(* Logix 5000 project; controller Celula_Envase_Automatica Emulate 5570 rev 32.11; software revision 32.03 *)

TASK MainTask (continuous, watchdog 500 ms) : MainProgram, Sequencer, Motor, IO
TASK PID_Task (periodic, rate 100 ms, priority 10, watchdog 500 ms) : PID_Control
TASK Simulation_Task (periodic, rate 100 ms, priority 11, watchdog 500 ms) : Process_Sim

MODULES
   Local : Emulate 5570 (ICP 2, rev 32.11)
END_MODULES

TYPE UDT_Cell :
STRUCT
   Cmd_Start : BOOL;   // Comando de partida da célula
   Cmd_Stop : BOOL;   // Comando de parada da célula
   Cmd_Reset : BOOL;   // Comando de reset de falhas
   AutoMode : BOOL;   // Seleção de modo automático
   Ready : BOOL;   // Célula pronta para operar
   Running : BOOL;   // Célula em operação
   Faulted : BOOL;   // Célula em falha
   State : DINT;   // Estado atual da sequência
   ProductionCount : DINT;   // Total de peças produzidas
   RejectCount : DINT;   // Total de peças rejeitadas
END_STRUCT
END_TYPE

TYPE UDT_Filling :
STRUCT
   Bottle_Present : BOOL;   // Indicação de garrafa presente na estação
   Fill_Cmd : BOOL;   // Comando de início do enchimento
   FillValve_Cmd : BOOL;   // Comando da válvula de enchimento
   Bottle_Volume : REAL;   // Volume atual da garrafa
   Target_Volume : REAL;   // Volume alvo de enchimento
   Filled : BOOL;   // Indicação de enchimento concluído
   Overfill : BOOL;   // Indicação de volume acima do limite
   Underfill : BOOL;   // Indicação de volume abaixo do limite
END_STRUCT
END_TYPE

TYPE UDT_Motor :
STRUCT
   Cmd_Start : BOOL;   // Comando de partida
   Cmd_Stop : BOOL;   // Comando de parada
   Enable : BOOL;   // Habilitação geral para operação do motor
   Reset : BOOL;   // Comando Reset
   Running : BOOL;   // Motor em funcionamento
   Stopped : BOOL;   // Motor parado
   Faulted : BOOL;   // Motor em falha
   Output : BOOL;   // Saida lógica de acionamento
   RunTime : DINT;   // Tempo acumulado de funcionamento
   StartCount : DINT;   // Quantidade de partidas
END_STRUCT
END_TYPE

TYPE UDT_PIDSim :
STRUCT
   PV : REAL;   // Variável de processo simulada
   SP : REAL;   // Setpoint da variável de processo
   CV : REAL;   // Saída de controle da malha PID
   Kp : REAL;   // Ganho proporcional da malha PID
   Ki : REAL;   // Ganho integral da malha PID
   Kd : REAL;   // Ganho derivativo da malha PID
   AutoMode : BOOL;   // Seleção do modo automático da malha PID
   ManualCV : REAL;   // Valor manual da saída de controle
END_STRUCT
END_TYPE

TYPE UDT_Tank :
STRUCT
   Level : REAL;   // Nível atual do tanque
   Level_SP : REAL;   // Setpoint de nível do tanque
   Inflow : REAL;   // Vazão de entrada no tanque
   Outflow : REAL;   // Vazão de saída do tanque
   ValveIn_Cmd : REAL;   // Comando de abertura da válvula de entrada
   ValveOut_Cmd : REAL;   // Comando de abertura da válvula de saída
   Mixer_Cmd : BOOL;   // Comando do agitador
   Mixer_Run : BOOL;   // Estado de operação do agitador
   High_Level : BOOL;   // Indicação de nível alto
   Low_Level : BOOL;   // Indicação de nível baixo
END_STRUCT
END_TYPE

ADD_ON_INSTRUCTION AOI_Motor   (* revision 1.0, vendor Lucas Larrosa *)
VAR_INPUT
   FaultInput : BOOL; {access None, required}
   Cmd_Start : BOOL; {required}
   Cmd_Stop : BOOL; {required}
   Enable : BOOL; {required}
   Reset : BOOL; {required}
END_VAR
VAR_OUTPUT
   Running : BOOL; {required}
   Stopped : BOOL; {required}
   Faulted : BOOL; {required}
   Output : BOOL; {required}
   RunTime : DINT; {required}
   StartCount : DINT; {required}
END_VAR

ROUTINE Logic   (* ladder *)
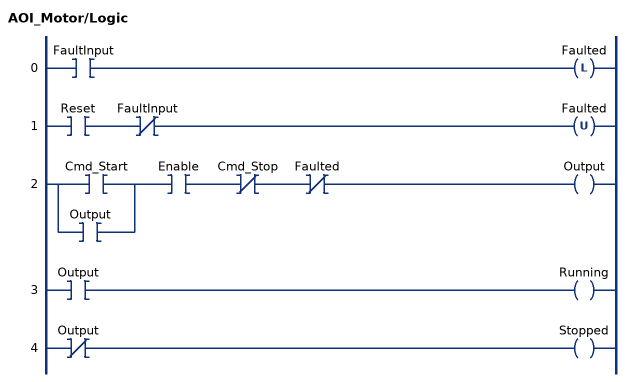
   0: XIC(FaultInput)OTL(Faulted);
   1: XIC(Reset)XIO(FaultInput)OTU(Faulted);
   2: [XIC(Cmd_Start) ,XIC(Output) ]XIC(Enable)XIO(Cmd_Stop)XIO(Faulted)OTE(Output);
   3: XIC(Output)OTE(Running);
   4: XIO(Output)OTE(Stopped);
END_ROUTINE
END_ADD_ON_INSTRUCTION

VAR_GLOBAL   (* controller tags *)
   aux_MotorStart : BOOL;
   aux_MotorStop : BOOL;
   aux_Ready : BOOL;
   aux_Running : BOOL;
   Cell01 : UDT_Cell := (Cmd_Start := 1, AutoMode := 1, State := 30, ProductionCount := 276, RejectCount := 55);
   ConveyorOut : BOOL;
   CycleComplete : BOOL;
   Data_ProductA_Pct : REAL;
   Data_ProductB_Pct : REAL;
   Enable_General : BOOL := 1;
   EStopOK : BOOL := 1;
   Fault_Motor01 : BOOL;
   Fill : BOOL := 1;
   Filling01 : UDT_Filling := (Fill_Cmd := 1, FillValve_Cmd := 1, Bottle_Volume := 9.799995, Target_Volume := 10.0);
   HMI_AutoMode : BOOL := 1;
   HMI_Reset : BOOL;
   HMI_Start : BOOL;
   HMI_Stop : BOOL;
   Inspect : BOOL;
   Inspection_Complete : BOOL;
   Inspection_OK : BOOL := 1;
   Motor01 : UDT_Motor := (Stopped := 1);
   Motor01_AutoCmd : BOOL;
   ONS_ProductionCount : BOOL;
   ONS_RejectCount : BOOL;
   PE_Entry : BOOL;
   PE_Exit : BOOL;
   PE_Inspection : BOOL;
   PID_Level : UDT_PIDSim;
   Reject : BOOL;
   Rejector_Command : BOOL;
   Rejector_Extended : BOOL;
   RejectReturn : BOOL;
   Stopped : BOOL;
   TankMix : UDT_Tank := (Level := 78.18737, Level_SP := 80.0, Inflow := 0.76456505, ValveIn_Cmd := 7.6456504);
   TankMix_LevelRate : REAL := 0.07645651;
   TankMix_NetFlow : REAL := 0.76456505;
   TankMix_SimDemand : DINT;
   TMR_RejectExtend : TIMER := (PRE := 500);
   TMR_RejectRetract : TIMER := (PRE := 500);
   TMR_SimConsumption : TIMER := (PRE := 30000, ACC := 15699, EN := 1, TT := 1);
   WaitPart : BOOL;
END_VAR

PROGRAM IO   (* main routine Main_IO *)
VAR
   InspectionCounter : DINT := 3;
   ONS_InspectionCount : BOOL;
   TMR_Inspection : TIMER := (PRE := 1500);
   TMR_PE_Entry : TIMER := (PRE := 1500);
   TMR_PE_Exit : TIMER := (PRE := 1500);
   TMR_PE_Inspection : TIMER := (PRE := 2000);
END_VAR

ROUTINE IO_Simulation   (* ladder *)
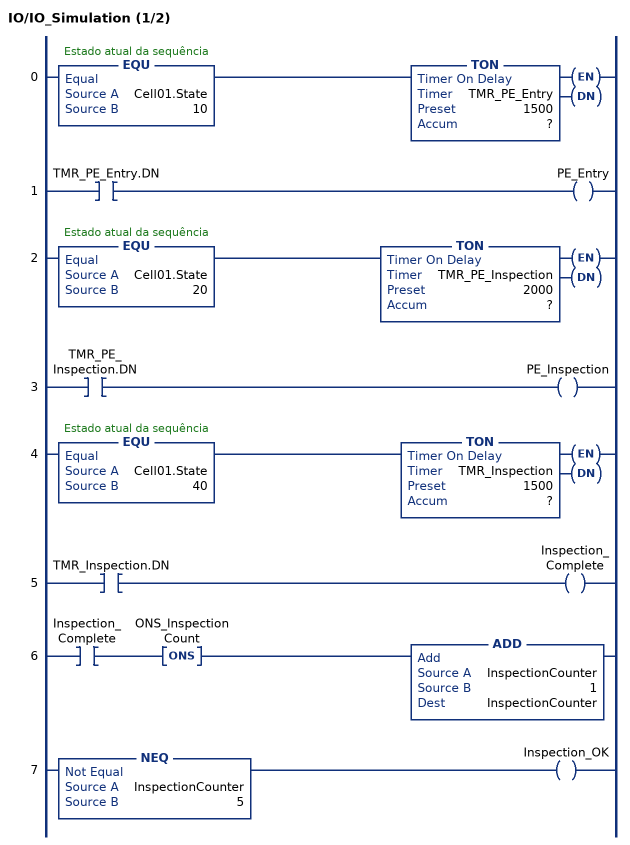
   0: EQU(Cell01.State,10)TON(TMR_PE_Entry,?,?);
   1: XIC(TMR_PE_Entry.DN)OTE(PE_Entry);
   2: EQU(Cell01.State,20)TON(TMR_PE_Inspection,?,?);
   3: XIC(TMR_PE_Inspection.DN)OTE(PE_Inspection);
   4: EQU(Cell01.State,40)TON(TMR_Inspection,?,?);
   5: XIC(TMR_Inspection.DN)OTE(Inspection_Complete);
   6: XIC(Inspection_Complete)ONS(ONS_InspectionCount)ADD(InspectionCounter,1,InspectionCounter);
   7: NEQ(InspectionCounter,5)OTE(Inspection_OK);
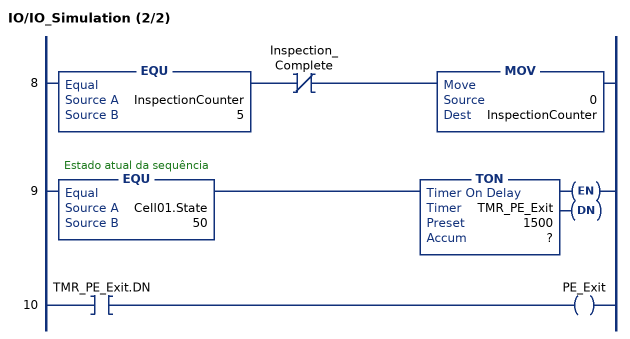
   8: EQU(InspectionCounter,5)XIO(Inspection_Complete)MOV(0,InspectionCounter);
   9: EQU(Cell01.State,50)TON(TMR_PE_Exit,?,?);
   10: XIC(TMR_PE_Exit.DN)OTE(PE_Exit);
END_ROUTINE

ROUTINE Main_IO   (* ladder *)
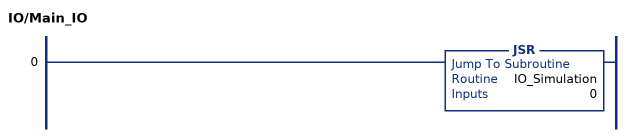
   0: JSR(IO_Simulation,0);
END_ROUTINE
END_PROGRAM

PROGRAM MainProgram   (* main routine MainRoutine *)

ROUTINE Main_Control   (* ladder *)
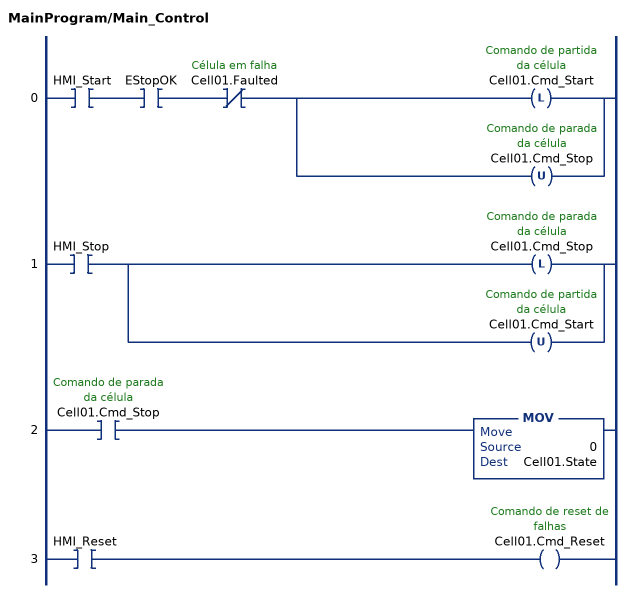
   0: XIC(HMI_Start)XIC(EStopOK)XIO(Cell01.Faulted)[OTL(Cell01.Cmd_Start) ,OTU(Cell01.Cmd_Stop) ];
   1: XIC(HMI_Stop)[OTL(Cell01.Cmd_Stop) ,OTU(Cell01.Cmd_Start) ];
   2: XIC(Cell01.Cmd_Stop)MOV(0,Cell01.State);
   3: XIC(HMI_Reset)OTE(Cell01.Cmd_Reset);
END_ROUTINE

ROUTINE Main_Interlocks   (* ladder *)
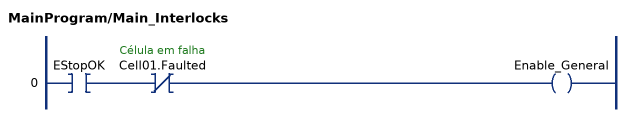
   0: XIC(EStopOK)XIO(Cell01.Faulted)OTE(Enable_General);
END_ROUTINE

ROUTINE Main_Status   (* ladder *)
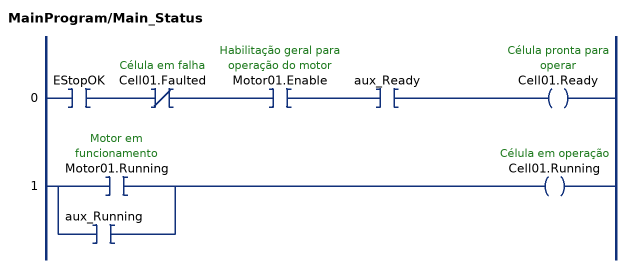
   0: XIC(EStopOK)XIO(Cell01.Faulted)XIC(Motor01.Enable)XIC(aux_Ready)OTE(Cell01.Ready);
   1: [XIC(Motor01.Running) ,XIC(aux_Running) ]OTE(Cell01.Running);
END_ROUTINE

ROUTINE MainRoutine   (* ladder *)
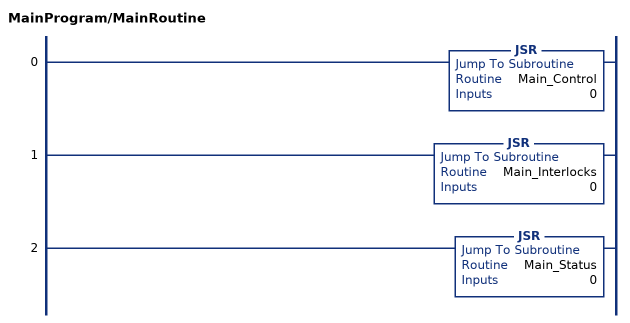
   0: JSR(Main_Control,0);
   1: JSR(Main_Interlocks,0);
   2: JSR(Main_Status,0);
END_ROUTINE
END_PROGRAM

PROGRAM Motor   (* main routine Main_Motor *)
VAR
   AOI_Motor01 : AOI_Motor := (Stopped := 1);
END_VAR

ROUTINE Main_Motor   (* ladder *)
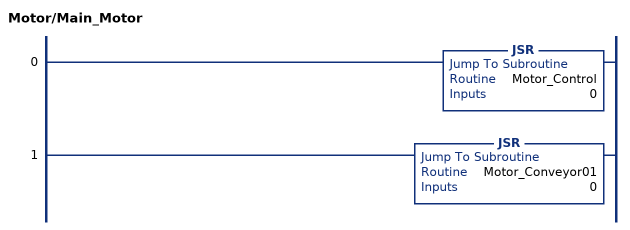
   0: JSR(Motor_Control,0);
   1: JSR(Motor_Conveyor01,0);
END_ROUTINE

ROUTINE Motor_Control   (* ladder *)
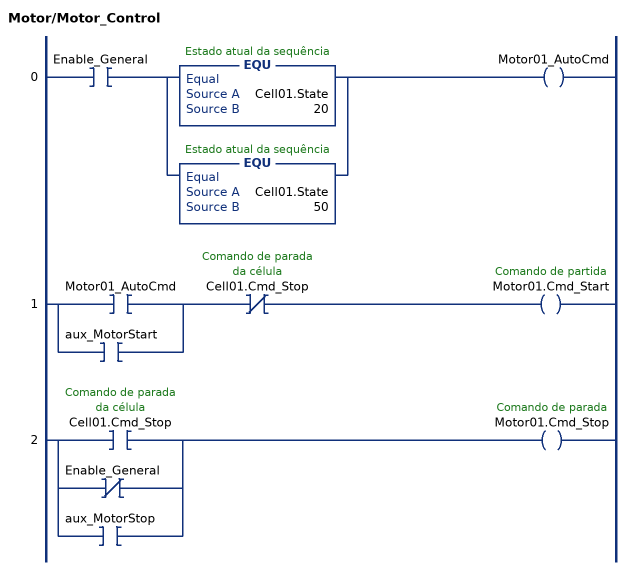
   0: XIC(Enable_General)[EQU(Cell01.State,20) ,EQU(Cell01.State,50) ]OTE(Motor01_AutoCmd);
   1: [XIC(Motor01_AutoCmd) ,XIC(aux_MotorStart) ]XIO(Cell01.Cmd_Stop)OTE(Motor01.Cmd_Start);
   2: [XIC(Cell01.Cmd_Stop) ,XIO(Enable_General) ,XIC(aux_MotorStop) ]OTE(Motor01.Cmd_Stop);
END_ROUTINE

ROUTINE Motor_Conveyor01   (* ladder *)
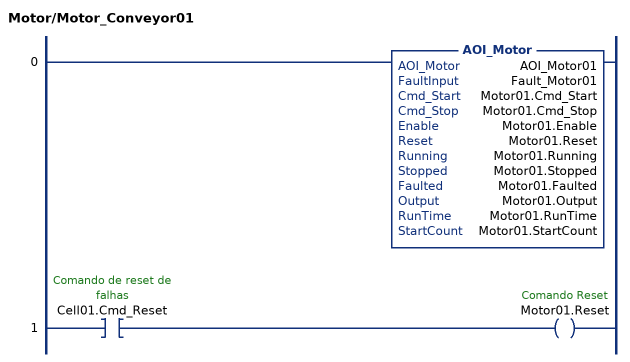
   0: AOI_Motor(AOI_Motor01,Fault_Motor01,Motor01.Cmd_Start,Motor01.Cmd_Stop,Motor01.Enable,Motor01.Reset,Motor01.Running,Motor01.Stopped,Motor01.Faulted,Motor01.Output,Motor01.RunTime,Motor01.StartCount);
   1: XIC(Cell01.Cmd_Reset)OTE(Motor01.Reset);
END_ROUTINE
END_PROGRAM

PROGRAM PID_Control   (* main routine Level_Control *)
VAR
   PIDE_01 : PID_ENHANCED := (PVEUMax := 100.0, SPHLimit := 100.0, RatioProg := 1.0, RatioOper := 1.0, RatioHLimit := 1.0, RatioLLimit := 1.0, CVEUMax := 100.0, CVHLimit := 100.0, PVEDerivative := 1, RTSTime := 1);
   PIDE_Level : PID_ENHANCED := (PV := 78.110916, PVEUMax := 100.0, SPProg := 80.0, SPOper := 80.0, SPHLimit := 100.0, RatioProg := 1.0, RatioOper := 1.0, RatioHLimit := 1.0, RatioLLimit := 1.0, CVOper := 7.6456504, CVEUMax := 100.0, CVHLimit := 100.0, PGain := 2.0, IGain := 0.15, PVEDerivative := 1, ProgProgReq := 1, ProgAutoReq := 1, RTSTime := 1, CVEU := 7.6456504, CV := 7.6456504, SP := 80.0, SPPercent := 80.0, PVPercent := 78.110916, E := 1.8890839, EPercent := 1.8890839, InitPrimary := 1, Ratio := 1.0, ProgOper := 1, Auto := 1, DeltaT := 0.1);   // Controlador PIDE de nível do tanque de mistura
END_VAR

ROUTINE Level_Control   (* function block diagram *)
   SHEET 1
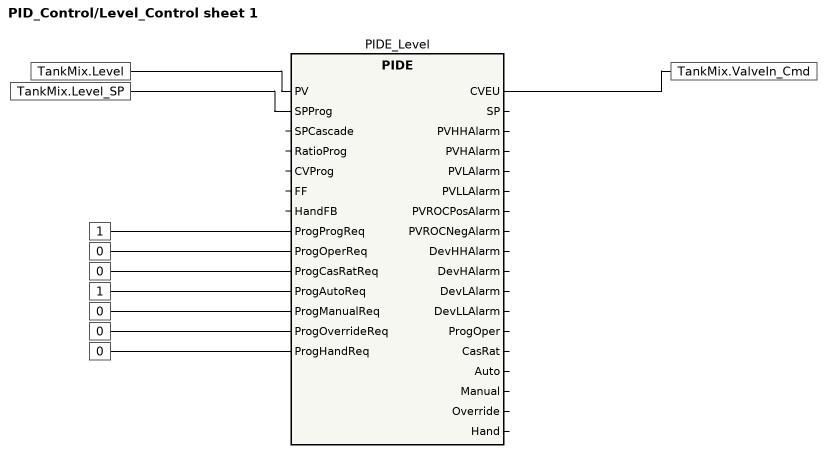
   PIDE_Level : PIDE(PV := TankMix.Level, SPProg := TankMix.Level_SP, ProgProgReq := 1, ProgOperReq := 0, ProgCasRatReq := 0, ProgAutoReq := 1, ProgManualReq := 0, ProgOverrideReq := 0, ProgHandReq := 0);   // unwired pins: SPCascade RatioProg CVProg FF HandFB SP PVHHAlarm PVHAlarm PVLAlarm PVLLAlarm PVROCPosAlarm PVROCNegAlarm DevHHAlarm DevHAlarm DevLAlarm DevLLAlarm ProgOper CasRat Auto Manual Override Hand
   TankMix.ValveIn_Cmd := PIDE_Level.CVEU;
END_ROUTINE
END_PROGRAM

PROGRAM Process_Sim   (* main routine Main_Process_Sim *)

ROUTINE Filling_Simulation   (* ladder *)
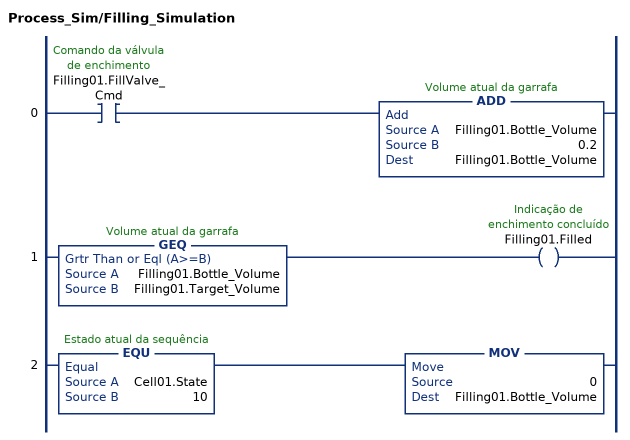
   0: XIC(Filling01.FillValve_Cmd)ADD(Filling01.Bottle_Volume,0.2,Filling01.Bottle_Volume);
   1: GEQ(Filling01.Bottle_Volume,Filling01.Target_Volume)OTE(Filling01.Filled);
   2: EQU(Cell01.State,10)MOV(0,Filling01.Bottle_Volume);
END_ROUTINE

ROUTINE Main_Process_Sim   (* ladder *)
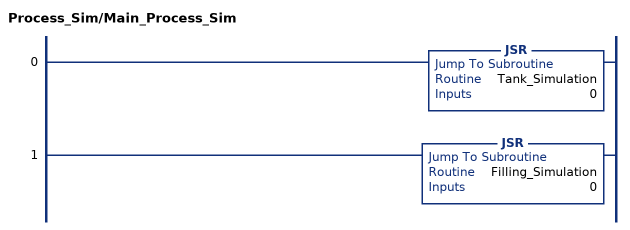
   0: JSR(Tank_Simulation,0);
   1: JSR(Filling_Simulation,0);
END_ROUTINE

ROUTINE Tank_Simulation   (* ladder *)
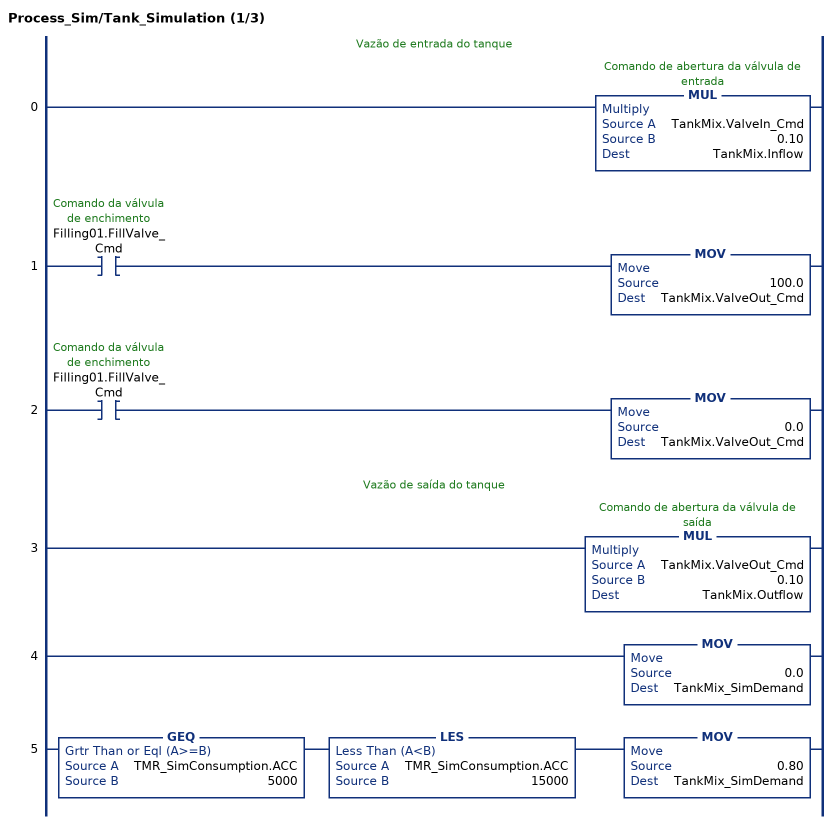
   // Vazão de entrada do tanque
   0: MUL(TankMix.ValveIn_Cmd,0.10,TankMix.Inflow);
   1: XIC(Filling01.FillValve_Cmd)MOV(100.0,TankMix.ValveOut_Cmd);
   2: XIC(Filling01.FillValve_Cmd)MOV(0.0,TankMix.ValveOut_Cmd);
   // Vazão de saída do tanque
   3: MUL(TankMix.ValveOut_Cmd,0.10,TankMix.Outflow);
   4: MOV(0.0,TankMix_SimDemand);
   5: GEQ(TMR_SimConsumption.ACC,5000)LES(TMR_SimConsumption.ACC,15000)MOV(0.80,TankMix_SimDemand);
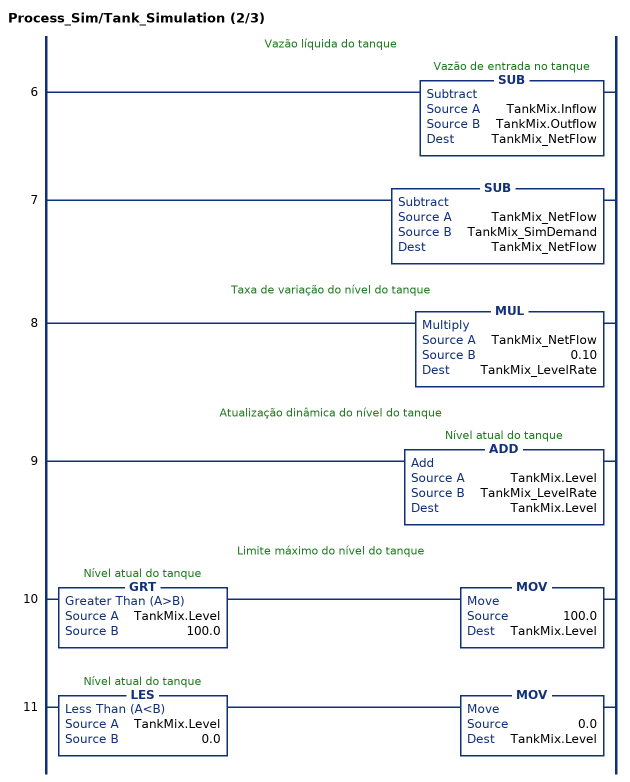
   // Vazão líquida do tanque
   6: SUB(TankMix.Inflow,TankMix.Outflow,TankMix_NetFlow);
   7: SUB(TankMix_NetFlow,TankMix_SimDemand,TankMix_NetFlow);
   // Taxa de variação do nível do tanque
   8: MUL(TankMix_NetFlow,0.10,TankMix_LevelRate);
   // Atualização dinâmica do nível do tanque
   9: ADD(TankMix.Level,TankMix_LevelRate,TankMix.Level);
   // Limite máximo do nível do tanque
   10: GRT(TankMix.Level,100.0)MOV(100.0,TankMix.Level);
   11: LES(TankMix.Level,0.0)MOV(0.0,TankMix.Level);
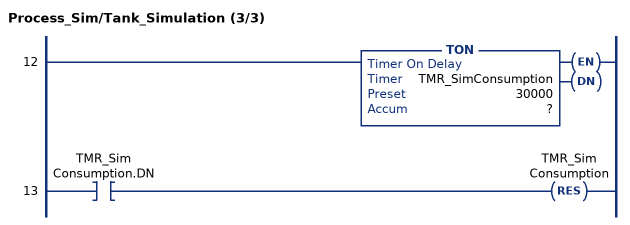
   12: TON(TMR_SimConsumption,?,?);
   13: XIC(TMR_SimConsumption.DN)RES(TMR_SimConsumption);
END_ROUTINE
END_PROGRAM

PROGRAM Sequencer   (* main routine Main_Sequencer *)
VAR
   STP_ConveyOut : SFC_STEP := (Status := 16#0820_0001, DN := 1, PauseTimer := 1, T := 1573, TMax := 2032, Count := 378);
   STP_ConveyToInspection : SFC_STEP := (Status := 16#0820_0001, DN := 1, PauseTimer := 1, T := 2067, TMax := 2087, Count := 473);
   STP_CycleComplete : SFC_STEP := (Status := 16#0820_0001, DN := 1, PauseTimer := 1, T := 21, TMax := 24, Count := 472);
   STP_Fill : SFC_STEP := (Status := 16#a820_0001, X := 1, SA := 1, DN := 1, PauseTimer := 1, T := 5241, TMax := 5492, Count := 473);
   STP_Inspect : SFC_STEP := (Status := 16#0820_0001, DN := 1, PauseTimer := 1, T := 1576, TMax := 1877, Count := 472);
   STP_Reject : SFC_STEP := (Status := 16#0820_0001, DN := 1, PauseTimer := 1, T := 544, TMax := 562, Count := 94);
   STP_RejectReturn : SFC_STEP := (Status := 16#0820_0001, DN := 1, PauseTimer := 1, T := 555, TMax := 565, Count := 94);
   STP_Stopped : SFC_STEP := (Status := 16#0820_0201, DN := 1, PauseTimer := 1, T := 22, TMax := 22, Count := 1);
   STP_WaitPart : SFC_STEP := (Status := 16#0820_0001, DN := 1, PauseTimer := 1, T := 1571, TMax := 1605, Count := 473);
   TR_AtInspection : BOOL := 1;
   TR_FillComplete : BOOL;
   TR_NewCycle : BOOL := 1;
   TR_PartDetected : BOOL := 1;
   TR_PartExited : BOOL := 1;
   TR_PartNOK : BOOL;
   TR_PartOK : BOOL := 1;
   TR_RejectExtended : BOOL := 1;
   TR_RejectRetracted : BOOL := 1;
   TR_StartCycle : BOOL := 1;
   Tran_000 : BOOL;
END_VAR

ROUTINE HMI_Sequencer   (* ladder *)
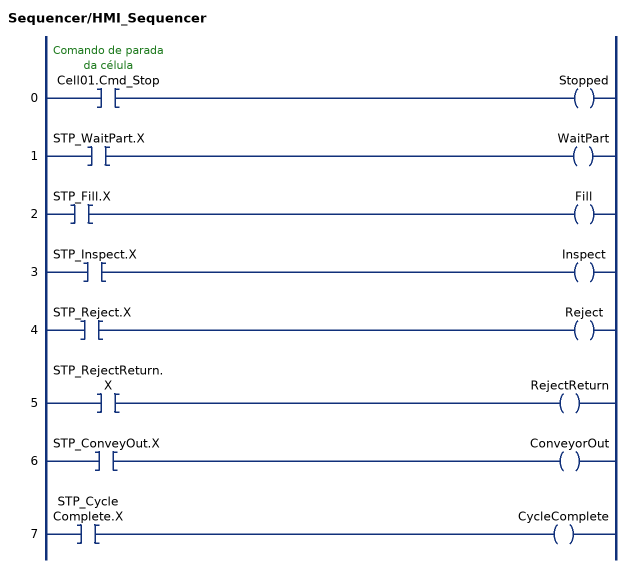
   0: XIC(Cell01.Cmd_Stop)OTE(Stopped);
   1: XIC(STP_WaitPart.X)OTE(WaitPart);
   2: XIC(STP_Fill.X)OTE(Fill);
   3: XIC(STP_Inspect.X)OTE(Inspect);
   4: XIC(STP_Reject.X)OTE(Reject);
   5: XIC(STP_RejectReturn.X)OTE(RejectReturn);
   6: XIC(STP_ConveyOut.X)OTE(ConveyorOut);
   7: XIC(STP_CycleComplete.X)OTE(CycleComplete);
END_ROUTINE

ROUTINE Main_Sequencer   (* ladder *)
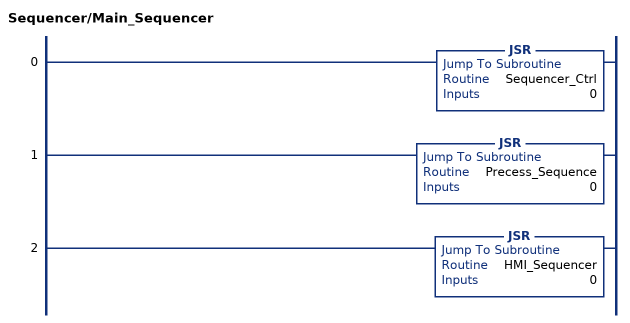
   0: JSR(Sequencer_Ctrl,0);
   1: JSR(Precess_Sequence,0);
   2: JSR(HMI_Sequencer,0);
END_ROUTINE

ROUTINE Precess_Sequence   (* sequential function chart *)
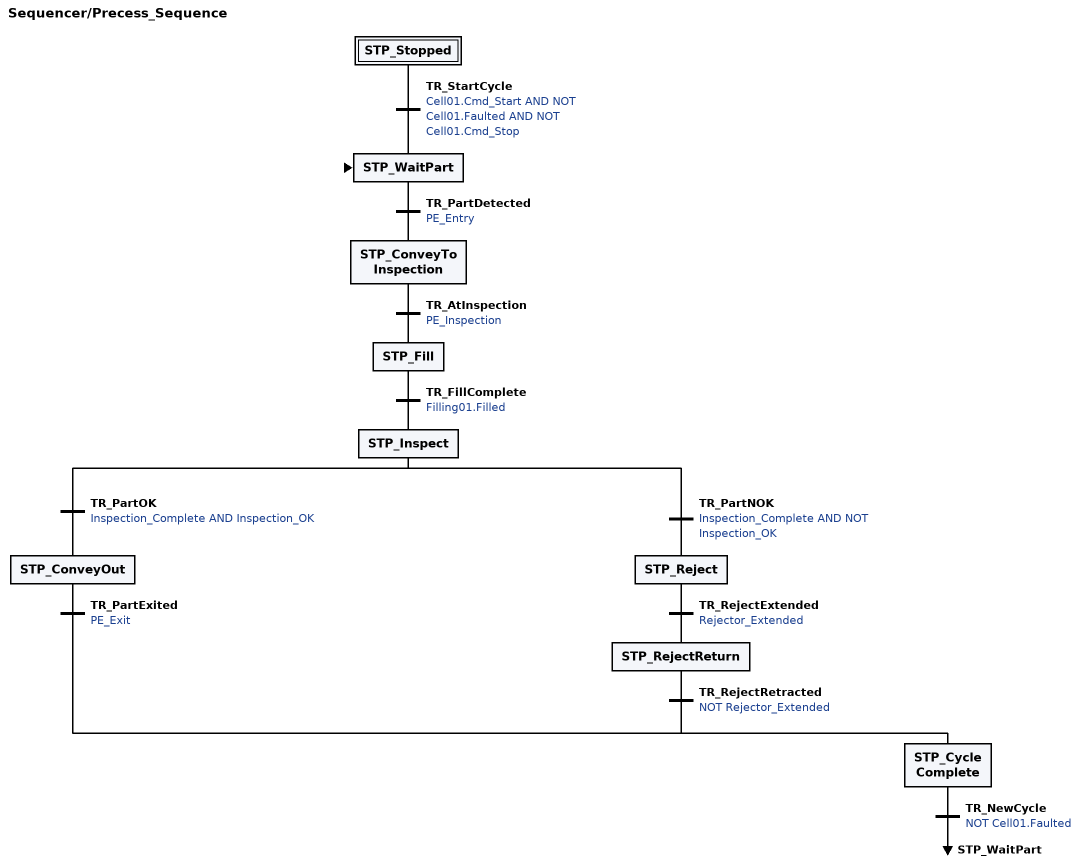
   INITIAL_STEP STP_Stopped:
   END_STEP
   TRANSITION TR_StartCycle FROM STP_Stopped TO STP_WaitPart
      := Cell01.Cmd_Start AND NOT Cell01.Faulted AND NOT Cell01.Cmd_Stop
   END_TRANSITION
   STEP STP_WaitPart:
   END_STEP
   TRANSITION TR_PartDetected FROM STP_WaitPart TO STP_ConveyToInspection
      := PE_Entry
   END_TRANSITION
   STEP STP_ConveyToInspection:
   END_STEP
   TRANSITION TR_AtInspection FROM STP_ConveyToInspection TO STP_Fill
      := PE_Inspection
   END_TRANSITION
   STEP STP_Fill:
   END_STEP
   TRANSITION TR_FillComplete FROM STP_Fill TO STP_Inspect
      := Filling01.Filled
   END_TRANSITION
   STEP STP_Inspect:
   END_STEP
   TRANSITION TR_PartOK FROM STP_Inspect TO STP_ConveyOut
      := Inspection_Complete AND Inspection_OK
   END_TRANSITION
   TRANSITION TR_PartNOK FROM STP_Inspect TO STP_Reject
      := Inspection_Complete AND NOT Inspection_OK
   END_TRANSITION
   STEP STP_ConveyOut:
   END_STEP
   STEP STP_Reject:
   END_STEP
   TRANSITION TR_PartExited FROM STP_ConveyOut TO STP_CycleComplete
      := PE_Exit
   END_TRANSITION
   TRANSITION TR_RejectExtended FROM STP_Reject TO STP_RejectReturn
      := Rejector_Extended
   END_TRANSITION
   STEP STP_RejectReturn:
   END_STEP
   TRANSITION TR_RejectRetracted FROM STP_RejectReturn TO STP_CycleComplete
      := NOT Rejector_Extended
   END_TRANSITION
   STEP STP_CycleComplete:
   END_STEP
   TRANSITION TR_NewCycle FROM STP_CycleComplete TO STP_WaitPart
      := NOT Cell01.Faulted
   END_TRANSITION
END_ROUTINE

ROUTINE Sequencer_Ctrl   (* ladder *)
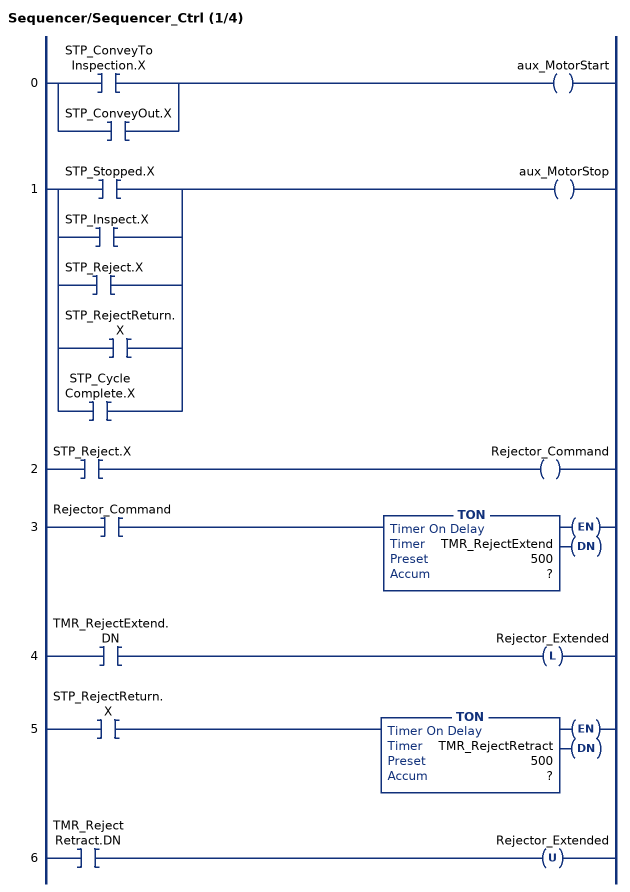
   0: [XIC(STP_ConveyToInspection.X) ,XIC(STP_ConveyOut.X) ]OTE(aux_MotorStart);
   1: [XIC(STP_Stopped.X) ,XIC(STP_Inspect.X) ,XIC(STP_Reject.X) ,XIC(STP_RejectReturn.X) ,XIC(STP_CycleComplete.X) ]OTE(aux_MotorStop);
   2: XIC(STP_Reject.X)OTE(Rejector_Command);
   3: XIC(Rejector_Command)TON(TMR_RejectExtend,?,?);
   4: XIC(TMR_RejectExtend.DN)OTL(Rejector_Extended);
   5: XIC(STP_RejectReturn.X)TON(TMR_RejectRetract,?,?);
   6: XIC(TMR_RejectRetract.DN)OTU(Rejector_Extended);
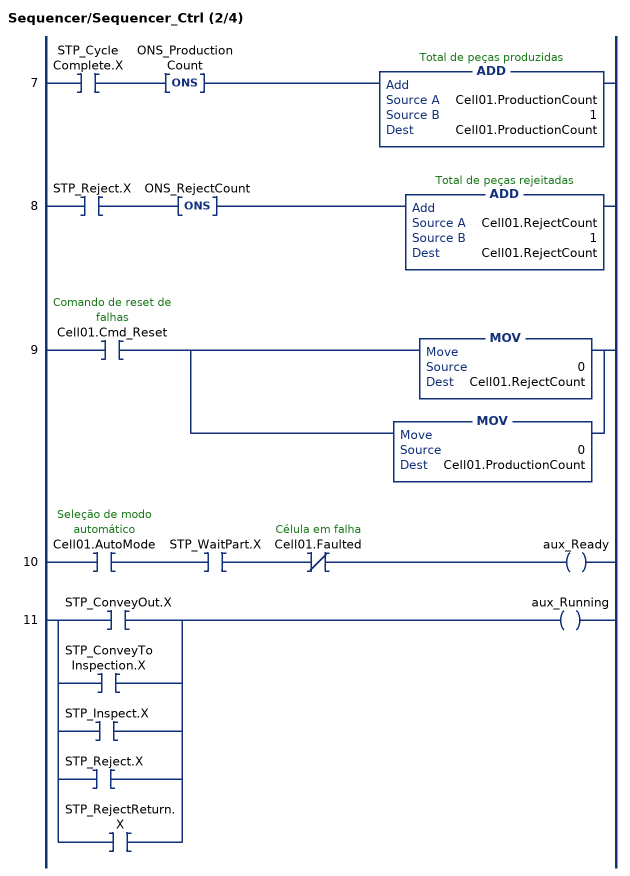
   7: XIC(STP_CycleComplete.X)ONS(ONS_ProductionCount)ADD(Cell01.ProductionCount,1,Cell01.ProductionCount);
   8: XIC(STP_Reject.X)ONS(ONS_RejectCount)ADD(Cell01.RejectCount,1,Cell01.RejectCount);
   9: XIC(Cell01.Cmd_Reset)[MOV(0,Cell01.RejectCount) ,MOV(0,Cell01.ProductionCount) ];
   10: XIC(Cell01.AutoMode)XIC(STP_WaitPart.X)XIO(Cell01.Faulted)OTE(aux_Ready);
   11: [XIC(STP_ConveyOut.X) ,XIC(STP_ConveyToInspection.X) ,XIC(STP_Inspect.X) ,XIC(STP_Reject.X) ,XIC(STP_RejectReturn.X) ]OTE(aux_Running);
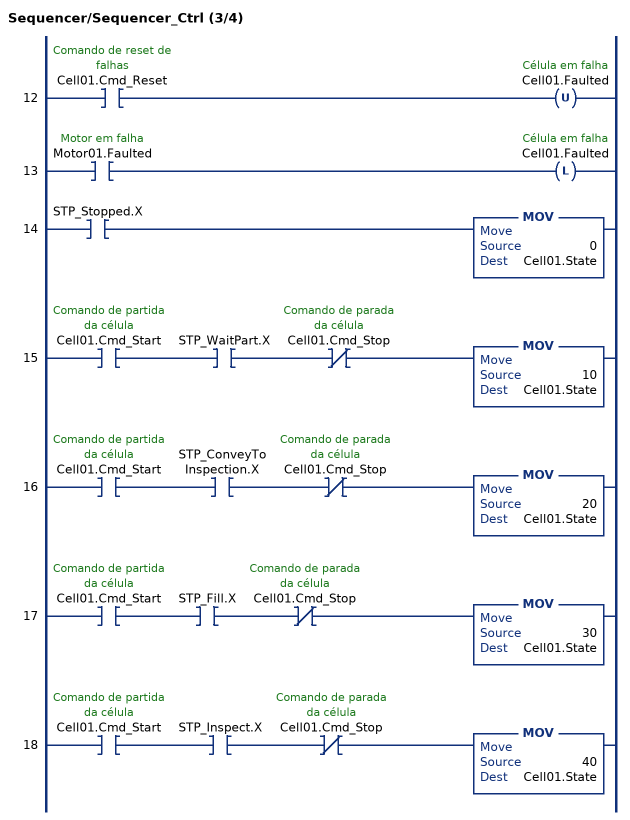
   12: XIC(Cell01.Cmd_Reset)OTU(Cell01.Faulted);
   13: XIC(Motor01.Faulted)OTL(Cell01.Faulted);
   14: XIC(STP_Stopped.X)MOV(0,Cell01.State);
   15: XIC(Cell01.Cmd_Start)XIC(STP_WaitPart.X)XIO(Cell01.Cmd_Stop)MOV(10,Cell01.State);
   16: XIC(Cell01.Cmd_Start)XIC(STP_ConveyToInspection.X)XIO(Cell01.Cmd_Stop)MOV(20,Cell01.State);
   17: XIC(Cell01.Cmd_Start)XIC(STP_Fill.X)XIO(Cell01.Cmd_Stop)MOV(30,Cell01.State);
   18: XIC(Cell01.Cmd_Start)XIC(STP_Inspect.X)XIO(Cell01.Cmd_Stop)MOV(40,Cell01.State);
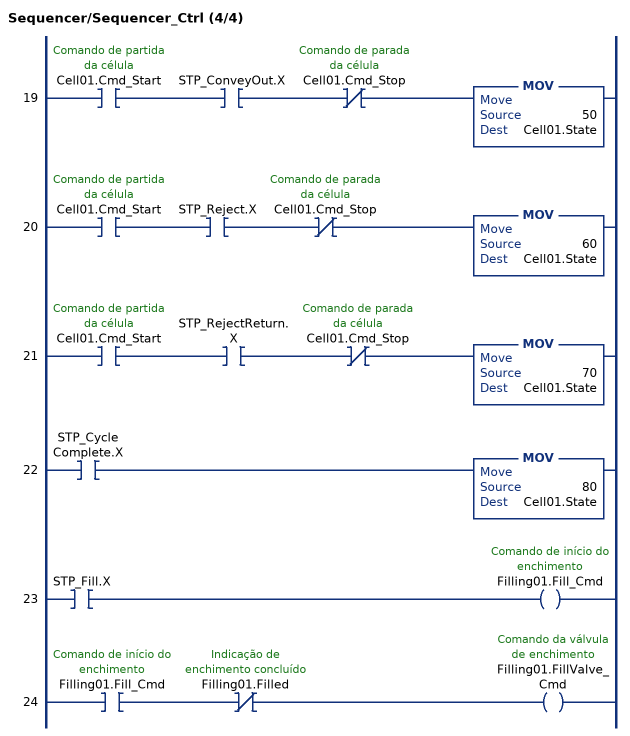
   19: XIC(Cell01.Cmd_Start)XIC(STP_ConveyOut.X)XIO(Cell01.Cmd_Stop)MOV(50,Cell01.State);
   20: XIC(Cell01.Cmd_Start)XIC(STP_Reject.X)XIO(Cell01.Cmd_Stop)MOV(60,Cell01.State);
   21: XIC(Cell01.Cmd_Start)XIC(STP_RejectReturn.X)XIO(Cell01.Cmd_Stop)MOV(70,Cell01.State);
   22: XIC(STP_CycleComplete.X)MOV(80,Cell01.State);
   23: XIC(STP_Fill.X)OTE(Filling01.Fill_Cmd);
   24: XIC(Filling01.Fill_Cmd)XIO(Filling01.Filled)OTE(Filling01.FillValve_Cmd);
END_ROUTINE
END_PROGRAM
